FUNCTION FC_DataFind : BOOL
VAR_INPUT
	WIDP : DINT;
	PmcData : POINTER TO DUT_St0Data;
	stPLCData : POINTER TO DUT_stPLCData;
	DataBuffer : POINTER TO DataBuffer;
END_VAR
VAR
	i : UINT;
END_VAR

FC_DataFind := FALSE;
IF WIDP > 0 THEN
	FOR i := 1 TO G.DATABUFFER_SIZE DO
		IF WIDP = DataBuffer[i].WIDP THEN
			PmcData^ := DataBuffer[i].PmcData;
			stPLCData^ := DataBuffer[i].stPLCData;
			FC_DataFind := TRUE;
			RETURN;
		END_IF
	END_FOR	
END_IF

END_FUNCTION

(* stored: Version 1.1.0.1, ProductVersion 3.1.4024.15
   POU FC_DataFind: Id {bf916154-5110-4f50-bf10-83eb694fe808}, SpecialFunc None *)
